Staubli VAL3: Record.pgx

public program Record(tool x_tTool)
  local string l_sString
  local num l_ni
  local num l_nVel
  local point l_pPoint
begin
  //
  wait(bRecord==true and !isEmpty())
  l_ni=1
  l_sString=""
  do
    l_nVel=getSpeed(x_tTool)
    l_pPoint=here(x_tTool,world)
    l_sString=toString("",l_ni)+" "+toString(".1",l_nVel)+" "+toString(".2", l_pPoint.trsf.x)+" "+toString(".2", l_pPoint.trsf.y)
    l_sString=l_sString+" "+toString(".2", l_pPoint.trsf.z)
    call WriteFile(l_sString)
    l_ni=l_ni+1
    delay(0)
  until isEmpty()==true
end
